// TIA Portal V20 export
DATA_BLOCK "CurrStroke"   // DB5
TITLE = Valori delle corse macchina attuali
{ S7_Optimized_Access := 'TRUE' }
// Sava i dati di valore Minimo e Massimo per gli assi correnti
// stored: MemoryReserve 100
   VAR
      Str : "Stroke";
   END_VAR
BEGIN
END_DATA_BLOCK
